Staubli VAL3: fileExit.pgx

program fileExit()
  local bool l_bRes
begin
  //
  l_bRes=$fileExists(sFileExist)
  if l_bRes
    gotoxy(1,7)
    put("文件存在:"+sFileExist)
  else
    gotoxy(1,7)
    put("文件不存在:"+sFileExist)
  endIf

end
